// Mitsubishi GX Works2 project: NAND2   PLC: Q03UDV

PROGRAM MAIN
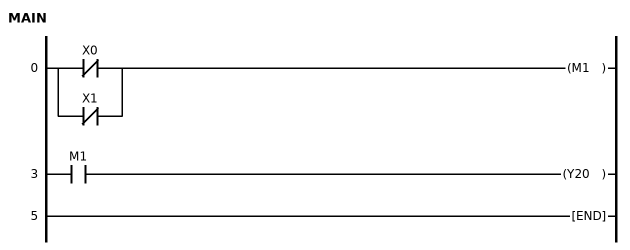
0     LDI     X0
      ORI     X1
      OUT     M1
3     LD      M1
      OUT     Y20
5     END
END_PROGRAM
